TYPE ST_AnnealingOvenSealingDefaultParameters :
STRUCT
	aSetPointLimitsTemperature : ARRAY[1..2] OF REAL := [30,40];
END_STRUCT
END_TYPE

(* stored: Version 1.1.0.1, ProductVersion 3.1.4024.10
   DUT ST_AnnealingOvenSealingDefaultParameters: Id {9ad3c7a9-2096-416c-8744-6995631add5f} *)
